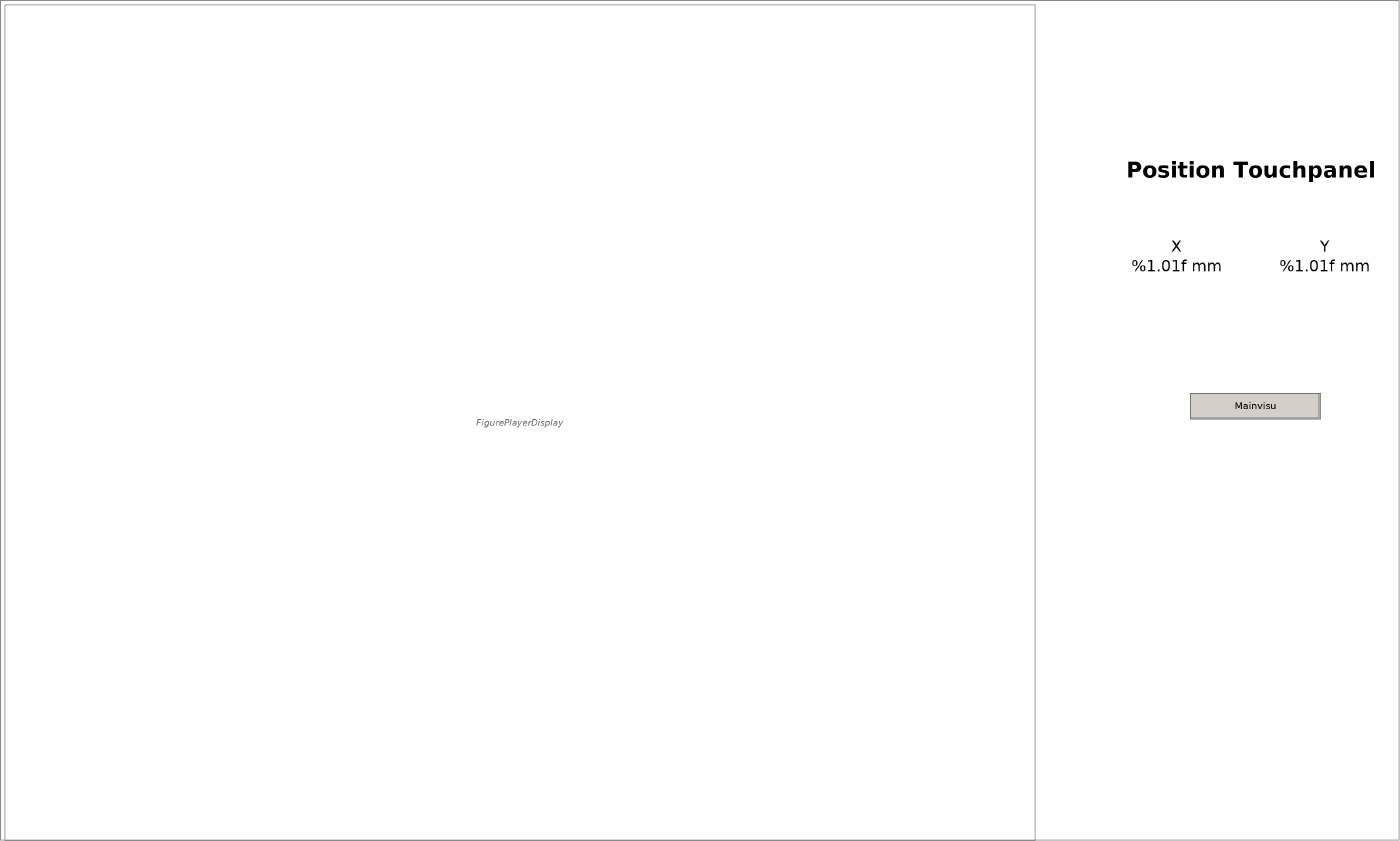
VISUALIZATION FigurePlayer  // 1608x967
    Rectangle (1436,269 171x51), "Y %1.01f mm", text variable: Touchpanel.touch_scale_y.rX_mm
    Rectangle (1266,269 171x51), "X %1.01f mm", text variable: Touchpanel.touch_scale_x.rX_mm
    Label (1266,165 342x60), "Position Touchpanel"
    Button (1367,452 150x30), "Mainvisu"
        OnMouseDown: change screen: Mainvisu
    Frame (5,5 1184x962)
        shows FigurePlayerDisplay()
END_VISUALIZATION

(* stored: Version 1.1.0.1, ProductVersion 3.1.4024.12
   Visu FigurePlayer: Id {af132e0e-c432-4516-b716-945794d96eeb} *)
